{attribute 'qualified_only'}
{attribute 'strict'}
{attribute 'to_string'} 

TYPE eDcLinkState :
(
	Disabled 	:= 0,
	Enabled	 	:= 1,
	Fault	 	:= 2
);
END_TYPE

(* stored: Version 1.1.0.1, ProductVersion 3.1.4026.18
   DUT eDcLinkState: Id {536ebfd8-c4ca-4029-ab35-bb84cc5c38f1} *)
